INTERFACE I_ActuatorFwdBwd EXTENDS I_ActuatorBase

{attribute 'monitoring' := 'call'}
PROPERTY public backwardStarted : BOOL
GET
END_GET
END_PROPERTY

{attribute 'monitoring' := 'call'}
PROPERTY public forwardStarted : BOOL
GET
END_GET
END_PROPERTY

METHOD public startBackward : BOOL
VAR_INPUT
END_VAR
END_METHOD

METHOD public startForward : BOOL
VAR_INPUT
END_VAR
END_METHOD

END_INTERFACE

(* stored: Version 1.1.0.1, ProductVersion 3.1.4024.3
   Itf I_ActuatorFwdBwd: Id {fdc28e6b-b113-4f5e-9504-a0f4634f1de3}
   Property backwardStarted: Id {01131f59-78b5-43b0-ac04-163ea79299f9}
   Get Get: Id {ca75166a-7cda-480a-94fe-1472b957eb4b}
   Property forwardStarted: Id {a1aaf5c2-a0d1-46c8-bcfb-7b04dd2ba8fd}
   Get Get: Id {698f3415-e0d5-4193-a76f-d2d00cafbe5b}
   Method startBackward: Id {d338b0d5-fb79-4592-88a4-6b0b315e8d0a}
   Method startForward: Id {8e24eae2-7369-45c7-ad34-ed1125182e1d} *)
